{region '#Template'}
	{attribute 'Version' := '1.0.0.0'}
	{attribute 'Tags' := '"LCID": "1031", "Text": "AC, Plant, AHU, Air handling unit"'}
	{attribute 'Tags' := '"LCID": "1033", "Text": "AC, Plant, AHU, Air handling unit"'}
	{attribute 'Description' := '"LCID": "1031", "Text": "Lüftungsanlage"'}
	{attribute 'Description' := '"LCID": "1033", "Text": "Air handling unit"'}
{endregion}
FUNCTION_BLOCK FB_BA_AHU_1St_PrHtr_ErcPl_Col EXTENDS FB_BA_View
VAR_INPUT CONSTANT	
	TOuA					: FB_BA_SensorAnalog_IO;			
	TExhA					: FB_BA_SensorAnalog_IO;	
	TSuA					: FB_BA_SensorAnalog_IO;	
	TExtA					: FB_BA_SensorAnalog_IO;								
	TRm						: FB_BA_SensorAnalog_IO;	
	DiffPrssOuAFilt			: FB_BA_SensorAnalog_IO;											
	FiltOuAMonit			: FB_BA_Hys_21;							
	DiffPrssExtAFilt		: FB_BA_SensorAnalog_IO;				
	FiltExtAMonit			: FB_BA_Hys_21;	
	SumNgtCol				: FB_BA_AC_SumNgtCol;	
	OpMod					: FB_BA_AC_OpMod1St;	
	OuADmp					: FB_BA_Dmp2P;	
	SuAPrss					: FB_BA_SensorAnalog_IO;	
	SuADiffPrss				: FB_BA_SensorAnalog_IO;		
	SuAFan					: FB_BA_MotCtlExt;	
	SuADiffPrssMonit		: FB_BA_FdbAnalog;								
	ExhADmp					: FB_BA_Dmp2P;	
	ExtAPrss				: FB_BA_SensorAnalog_IO;	
	ExtADiffPrss			: FB_BA_SensorAnalog_IO;		
	ExtAFan					: FB_BA_MotCtlExt;								
	ExtADiffPrssMonit		: FB_BA_FdbAnalog;
	SpTRm					: FB_BA_AC_SpTRm_01;	
	TCasCtrl				: FB_BA_AC_TCasCtrl_01;										 								
	TSeqLink				: FB_BA_SequenceLink;
	PreHtr					: FB_BA_AC_PreHtr;	
	Erc						: FB_BA_AC_ErcPl_02;								
	Col						: FB_BA_AC_ColT_02;								
	PlantCtrl				: FB_BA_PlantCtrl;							
	GeneralSettings			: FB_BA_RawSubscriber;
	stGeneralSettings		: ST_BA_GeneralSettings;
END_VAR	
VAR
	PlantLock				: FB_BA_PlantLock	:= (iParent := THIS^);	
	
	PlantControlStatus   	:FB_BA_Label2x :=(iAggregate:=LblControl_PlantControl,		iFunction:=LblFunctions_Status);
	TSequenceControlStatus  :FB_BA_Label2x :=(iAggregate:=LblControl_TSequenceControl,	iFunction:=LblFunctions_Status);	
END_VAR
VAR // added by the converter: edge detectors and wires of the graphical bodies
    _w1 : ANY;
END_VAR

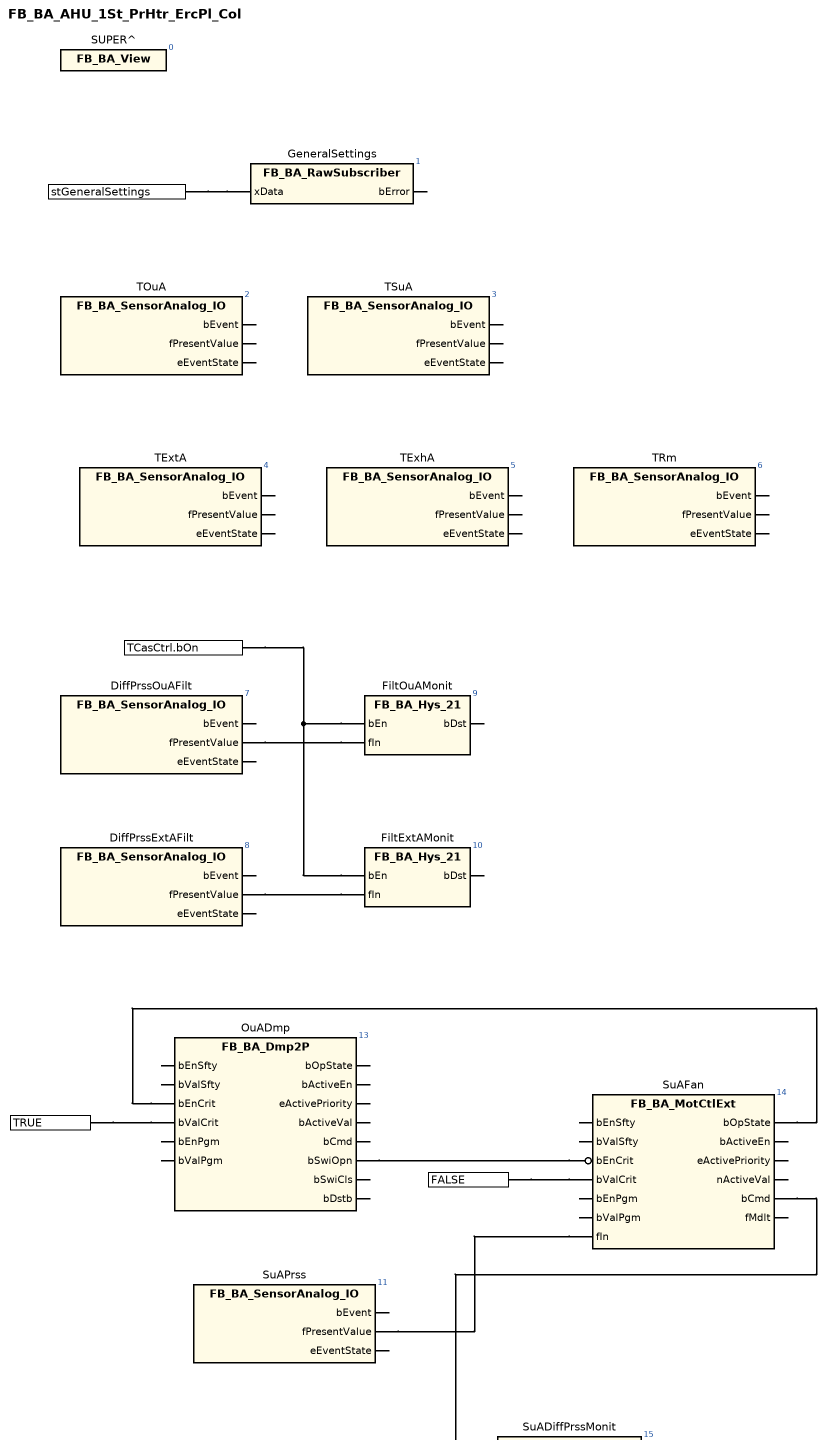
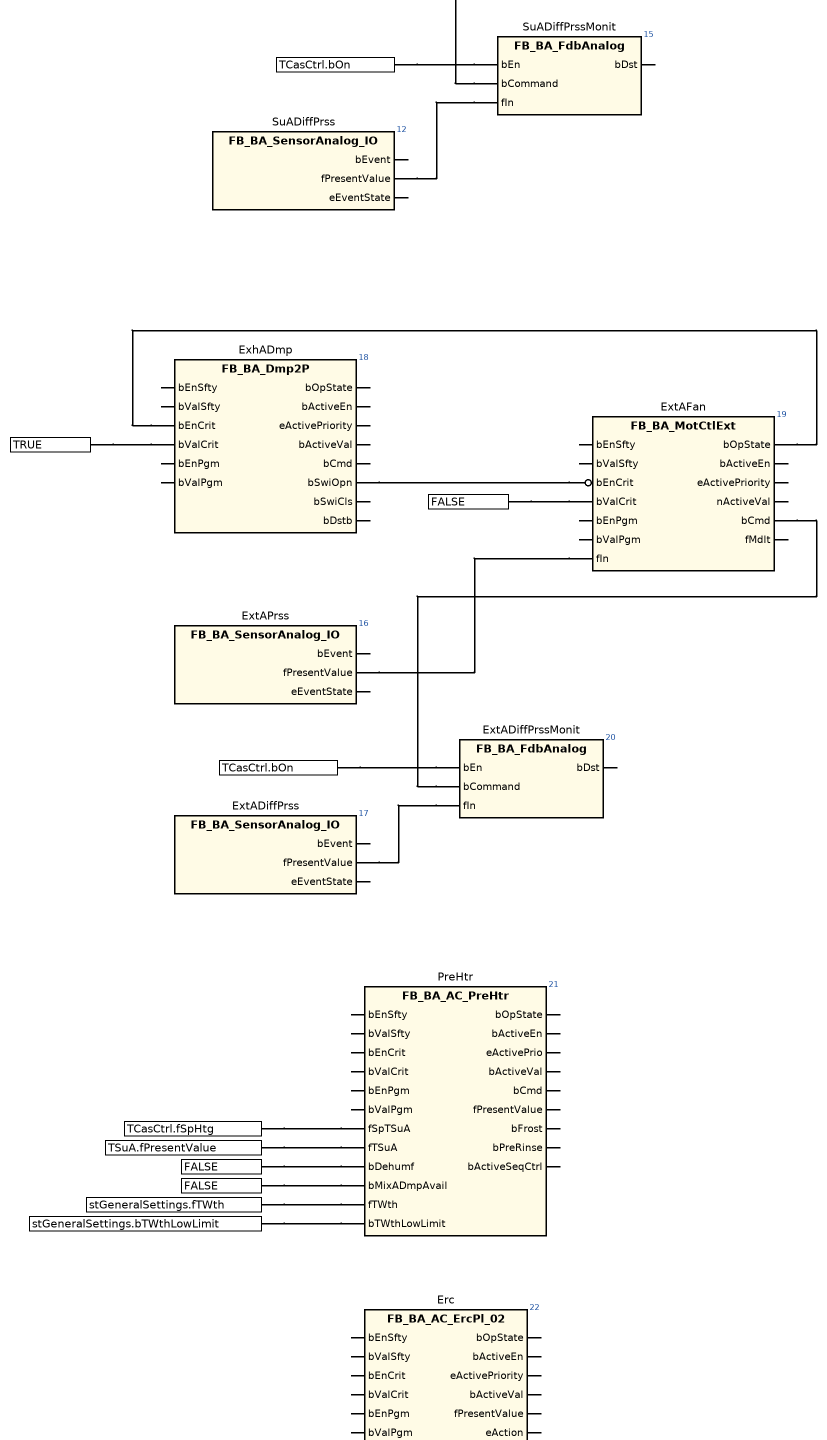
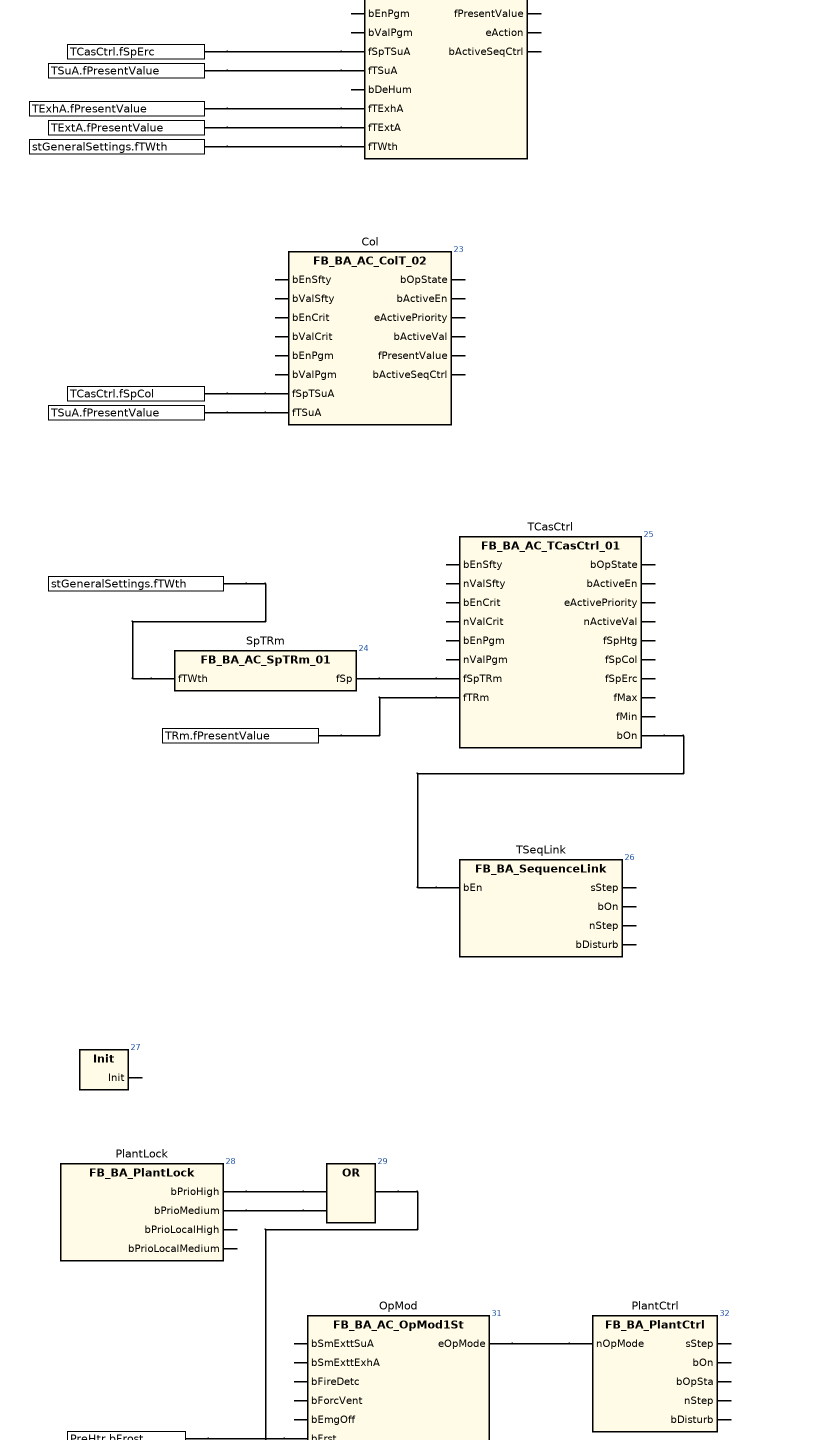
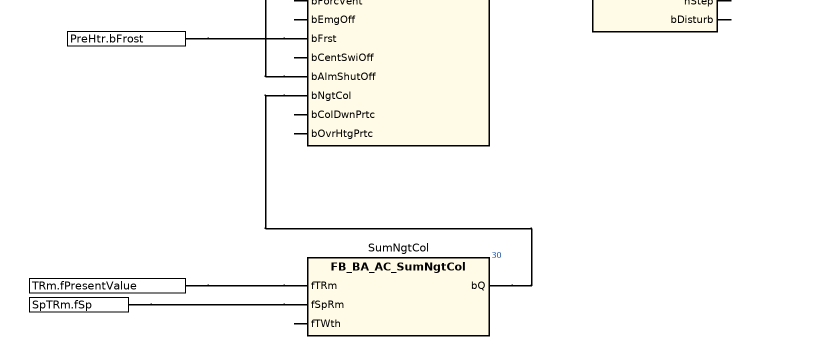
SUPER^(); // FB_BA_View
GeneralSettings(xData := stGeneralSettings); // FB_BA_RawSubscriber
TOuA(); // FB_BA_SensorAnalog_IO
TSuA(); // FB_BA_SensorAnalog_IO
TExtA(); // FB_BA_SensorAnalog_IO
TExhA(); // FB_BA_SensorAnalog_IO
TRm(); // FB_BA_SensorAnalog_IO
DiffPrssOuAFilt(); // FB_BA_SensorAnalog_IO
DiffPrssExtAFilt(); // FB_BA_SensorAnalog_IO
FiltOuAMonit(bEn := TCasCtrl.bOn, fIn := DiffPrssOuAFilt.fPresentValue); // FB_BA_Hys_21
FiltExtAMonit(bEn := TCasCtrl.bOn, fIn := DiffPrssExtAFilt.fPresentValue); // FB_BA_Hys_21
SuAPrss(); // FB_BA_SensorAnalog_IO
SuADiffPrss(); // FB_BA_SensorAnalog_IO
OuADmp(bEnCrit := SuAFan.bOpState, bValCrit := TRUE); // FB_BA_Dmp2P
SuAFan(bEnCrit := NOT OuADmp.bSwiOpn, bValCrit := FALSE, fIn := SuAPrss.fPresentValue); // FB_BA_MotCtlExt
SuADiffPrssMonit(bEn := TCasCtrl.bOn, bCommand := SuAFan.bCmd, fIn := SuADiffPrss.fPresentValue); // FB_BA_FdbAnalog
ExtAPrss(); // FB_BA_SensorAnalog_IO
ExtADiffPrss(); // FB_BA_SensorAnalog_IO
ExhADmp(bEnCrit := ExtAFan.bOpState, bValCrit := TRUE); // FB_BA_Dmp2P
ExtAFan(bEnCrit := NOT ExhADmp.bSwiOpn, bValCrit := FALSE, fIn := ExtAPrss.fPresentValue); // FB_BA_MotCtlExt
ExtADiffPrssMonit(bEn := TCasCtrl.bOn, bCommand := ExtAFan.bCmd, fIn := ExtADiffPrss.fPresentValue); // FB_BA_FdbAnalog
PreHtr(
    fSpTSuA := TCasCtrl.fSpHtg,
    fTSuA := TSuA.fPresentValue,
    bDehumf := FALSE,
    bMixADmpAvail := FALSE,
    fTWth := stGeneralSettings.fTWth,
    bTWthLowLimit := stGeneralSettings.bTWthLowLimit); // FB_BA_AC_PreHtr
Erc(
    fSpTSuA := TCasCtrl.fSpErc,
    fTSuA := TSuA.fPresentValue,
    fTExhA := TExhA.fPresentValue,
    fTExtA := TExtA.fPresentValue,
    fTWth := stGeneralSettings.fTWth); // FB_BA_AC_ErcPl_02
Col(fSpTSuA := TCasCtrl.fSpCol, fTSuA := TSuA.fPresentValue); // FB_BA_AC_ColT_02
SpTRm(fTWth := stGeneralSettings.fTWth); // FB_BA_AC_SpTRm_01
TCasCtrl(fSpTRm := SpTRm.fSp, fTRm := TRm.fPresentValue); // FB_BA_AC_TCasCtrl_01
TSeqLink(bEn := TCasCtrl.bOn); // FB_BA_SequenceLink
Init();
PlantLock(); // FB_BA_PlantLock
_w1 := PlantLock.bPrioHigh OR PlantLock.bPrioMedium;
SumNgtCol(fTRm := TRm.fPresentValue, fSpRm := SpTRm.fSp); // FB_BA_AC_SumNgtCol
OpMod(bFrst := PreHtr.bFrost, bAlmShutOff := _w1, bNgtCol := SumNgtCol.bQ); // FB_BA_AC_OpMod1St
PlantCtrl(nOpMode := OpMod.eOpMode); // FB_BA_PlantCtrl

METHOD FB_init : BOOL
VAR_INPUT
	bInitRetains : BOOL; // if TRUE, the retain variables are initialized (warm start / cold start)
	bInCopyCode : BOOL;  // if TRUE, the instance afterwards gets moved into the copy code (online change)
END_VAR
TOuA.iParent								:= THIS^;		
TOuA.iLabel 								:= LblCmpAC.AHU_TOuA;	
TOuA.sObjectName							:= '{Idx=01}';	
TOuA.eDPADMode								:= E_BA_DPADMode.eInclude;										
TOuA.MV.eUnit								:= E_BA_Unit.eTemperature_DegreesCelsius;
TOuA.MV.fResolution 						:= 0.01;
TOuA.MV.fScaleOffset 						:= 0; 
TOuA.MV.eEnPlantLock						:= E_BA_LockPriority.eNoLock;

TExhA.iParent								:= THIS^;		
TExhA.iLabel 								:= LblCmpAC.AHU_TExhA;	
TExhA.sObjectName							:= '{Idx=01}';												
TExhA.eDPADMode								:= E_BA_DPADMode.eInclude;										
TExhA.MV.eUnit								:= E_BA_Unit.eTemperature_DegreesCelsius;
TExhA.MV.fResolution 						:= 0.01;
TExhA.MV.fScaleOffset 						:= 0; 
TExhA.MV.eEnPlantLock						:= E_BA_LockPriority.eNoLock;

TSuA.iParent								:= THIS^;		
TSuA.iLabel 								:= LblCmpAC.AHU_TSuA;	
TSuA.sObjectName							:= '{Idx=01}';
TSuA.eDPADMode								:= E_BA_DPADMode.eInclude;										
TSuA.MV.eUnit								:= E_BA_Unit.eTemperature_DegreesCelsius;
TSuA.MV.fResolution 						:= 0.01;
TSuA.MV.fScaleOffset 						:= 0; 
TSuA.MV.eEnPlantLock						:= E_BA_LockPriority.eMedium;

TExtA.iParent								:= THIS^;
TExtA.iLabel 								:= LblCmpAC.AHU_TExtA;	
TExtA.sObjectName							:= '{Idx=01}'; 
TExtA.eDPADMode								:= E_BA_DPADMode.eInclude;										
TExtA.MV.eUnit								:= E_BA_Unit.eTemperature_DegreesCelsius;
TExtA.MV.fResolution 						:= 0.01;
TExtA.MV.fScaleOffset 						:= 0; 
TExtA.MV.eEnPlantLock						:= E_BA_LockPriority.eNoLock;

TRm.iParent									:= THIS^;		
TRm.iLabel 									:= LblCmpAC.AHU_TRm;	
TRm.sObjectName								:= '{Idx=01}';
TRm.eDPADMode								:= E_BA_DPADMode.eInclude;										
TRm.MV.eUnit								:= E_BA_Unit.eTemperature_DegreesCelsius;
TRm.MV.fResolution 							:= 0.01;
TRm.MV.fScaleOffset 						:= 0;
TRm.MV.eEnPlantLock							:= E_BA_LockPriority.eNoLock;

DiffPrssOuAFilt.iParent						:= THIS^;		
DiffPrssOuAFilt.iLabel 						:= LblCmpAC.AHU_DiffPrssOuAFilt;	
DiffPrssOuAFilt.sObjectName					:= '{Idx=03}';												
DiffPrssOuAFilt.eDPADMode					:= E_BA_DPADMode.eInclude;										
DiffPrssOuAFilt.MV.eUnit					:= E_BA_Unit.ePressure_Pascals;
DiffPrssOuAFilt.MV.fResolution 				:= 0.03051851;
DiffPrssOuAFilt.MV.fScaleOffset 			:= 0; 
DiffPrssOuAFilt.MV.eEnPlantLock				:= E_BA_LockPriority.eNoLock;

FiltOuAMonit.iParent						:= THIS^;
FiltOuAMonit.iLabel							:= LblCmpAC.AHU_FiltOuAMonit;
FiltOuAMonit.sObjectName					:= '{Idx=01}';										 
FiltOuAMonit.eDPADMode						:= E_BA_DPADMode.eInclude;
FiltOuAMonit.DstPreAlarm.eEnPlantLock		:= E_BA_LockPriority.eNoLock;	
FiltOuAMonit.DstMainAlarm.eEnPlantLock		:= E_BA_LockPriority.eMedium;

DiffPrssExtAFilt.iParent					:= THIS^;		
DiffPrssExtAFilt.iLabel 					:= LblCmpAC.AHU_DiffPrssExtAFilt;	
DiffPrssExtAFilt.sObjectName				:= '{Idx=04}';
DiffPrssExtAFilt.eDPADMode					:= E_BA_DPADMode.eInclude;										
DiffPrssExtAFilt.MV.eUnit					:= E_BA_Unit.ePressure_Pascals;
DiffPrssExtAFilt.MV.fResolution 			:= 0.03051851;
DiffPrssExtAFilt.MV.fScaleOffset 			:= 0; 
DiffPrssExtAFilt.MV.eEnPlantLock			:= E_BA_LockPriority.eNoLock;

FiltExtAMonit.iParent						:= THIS^;
FiltExtAMonit.iLabel						:= LblCmpAC.AHU_FiltExtAMonit;
FiltExtAMonit.sObjectName					:= '{Idx=02}';										 
FiltExtAMonit.eDPADMode						:= E_BA_DPADMode.eInclude;
FiltExtAMonit.DstPreAlarm.eEnPlantLock		:= E_BA_LockPriority.eNoLock;	
FiltExtAMonit.DstMainAlarm.eEnPlantLock		:= E_BA_LockPriority.eMedium;

SumNgtCol.iParent							:= THIS^;
SumNgtCol.iLabel							:= LblCmpAC.AHU_SumNgtCol;
SumNgtCol.sObjectName						:= '{Idx=01}';										 
SumNgtCol.eDPADMode							:= E_BA_DPADMode.eInclude;								

OpMod.iParent								:= THIS^;
OpMod.iLabel								:= LblCmpAC.AHU_OpMod;
OpMod.sObjectName							:= '{Idx=01}';										 
OpMod.eDPADMode								:= E_BA_DPADMode.eInclude;								

OuADmp.iParent								:= THIS^;
OuADmp.iLabel								:= LblCmpAC.AHU_OuADmp;
OuADmp.sObjectName							:= '{Idx=01}';										 
OuADmp.eDPADMode							:= E_BA_DPADMode.eInclude;
OuADmp.MonitOpen.Dst.eEnPlantLock			:= E_BA_LockPriority.eLocalMedium;								
OuADmp.MonitClose.Dst.eEnPlantLock			:= E_BA_LockPriority.eNoLock;								

SuAPrss.iParent								:= THIS^;		
SuAPrss.iLabel 								:= LblCmpAC.AHU_SuAPrss;	
SuAPrss.sObjectName							:= '{Idx=01}';
SuAPrss.eDPADMode							:= E_BA_DPADMode.eInclude;																						
SuAPrss.MV.eUnit							:= E_BA_Unit.ePressure_Pascals;
SuAPrss.MV.fResolution 						:= 0.03051851;
SuAPrss.MV.fScaleOffset 					:= 0;
SuAPrss.MV.eEnPlantLock						:= E_BA_LockPriority.eNoLock;

SuADiffPrss.iParent							:= THIS^;		
SuADiffPrss.iLabel 							:= LblCmpAC.AHU_SuADiffPrss;	
SuADiffPrss.sObjectName						:= '{Idx=01}';
SuADiffPrss.eDPADMode						:= E_BA_DPADMode.eInclude;																						
SuADiffPrss.MV.eUnit						:= E_BA_Unit.ePressure_Pascals;
SuADiffPrss.MV.fResolution 					:= 0.03051851;
SuADiffPrss.MV.fScaleOffset 				:= 0; 
SuADiffPrss.MV.eEnPlantLock					:= E_BA_LockPriority.eNoLock;

SuAFan.iParent								:= THIS^;
SuAFan.iLabel								:= LblCmpAC.AHU_SuAFan;
SuAFan.sObjectName							:= '{Idx=01}';										 
SuAFan.eDPADMode							:= E_BA_DPADMode.eInclude;								
SuAFan.Dst.eEnPlantLock						:= E_BA_LockPriority.eMedium;
SuAFan.ThOvrld.eEnPlantLock					:= E_BA_LockPriority.eMedium;	
SuAFan.MntnSwi.eEnPlantLock					:= E_BA_LockPriority.eMedium;

SuADiffPrssMonit.iParent					:= THIS^;
SuADiffPrssMonit.iLabel						:= LblCmpAC.AHU_SuADiffPrssMonit;
SuADiffPrssMonit.sObjectName				:= '{Idx=01}';										 
SuADiffPrssMonit.eDPADMode					:= E_BA_DPADMode.eInclude;								
SuADiffPrssMonit.Dst.eEnPlantLock			:= E_BA_LockPriority.eMedium;										

ExhADmp.iParent								:= THIS^;
ExhADmp.iLabel								:= LblCmpAC.AHU_ExhADmp;
ExhADmp.sObjectName							:= '{Idx=02}';										 
ExhADmp.eDPADMode							:= E_BA_DPADMode.eInclude;								
ExhADmp.MonitOpen.Dst.eEnPlantLock			:= E_BA_LockPriority.eLocalMedium;								
ExhADmp.MonitClose.Dst.eEnPlantLock			:= E_BA_LockPriority.eNoLock;				

ExtAPrss.iParent							:= THIS^;		
ExtAPrss.iLabel 							:= LblCmpAC.AHU_ExtAPrss;	
ExtAPrss.sObjectName						:= '{Idx=01}';												
ExtAPrss.eDPADMode							:= E_BA_DPADMode.eInclude;																						
ExtAPrss.MV.eUnit							:= E_BA_Unit.ePressure_Pascals;
ExtAPrss.MV.fResolution 					:= 0.03051851;
ExtAPrss.MV.fScaleOffset 					:= 0; 
ExtAPrss.MV.eEnPlantLock					:= E_BA_LockPriority.eNoLock;

ExtADiffPrss.iParent						:= THIS^;		
ExtADiffPrss.iLabel 						:= LblCmpAC.AHU_ExtADiffPrss;	
ExtADiffPrss.sObjectName					:= '{Idx=02}';
ExtADiffPrss.eDPADMode						:= E_BA_DPADMode.eInclude;																						
ExtADiffPrss.MV.eUnit						:= E_BA_Unit.ePressure_Pascals;
ExtADiffPrss.MV.fResolution 				:= 0.03051851;
ExtADiffPrss.MV.fScaleOffset 				:= 0; 
ExtADiffPrss.MV.eEnPlantLock				:= E_BA_LockPriority.eNoLock;

ExtAFan.iParent								:= THIS^;
ExtAFan.iLabel								:= LblCmpAC.AHU_ExtAFan;
ExtAFan.sObjectName							:= '{Idx=01}';										 
ExtAFan.eDPADMode							:= E_BA_DPADMode.eInclude;								
ExtAFan.Dst.eEnPlantLock					:= E_BA_LockPriority.eMedium;
ExtAFan.ThOvrld.eEnPlantLock				:= E_BA_LockPriority.eMedium;	
ExtAFan.MntnSwi.eEnPlantLock				:= E_BA_LockPriority.eMedium;

ExtADiffPrssMonit.iParent					:= THIS^;
ExtADiffPrssMonit.iLabel					:= LblCmpAC.AHU_ExtADiffPrssMonit;
ExtADiffPrssMonit.sObjectName				:= '{Idx=02}';										 
ExtADiffPrssMonit.eDPADMode					:= E_BA_DPADMode.eInclude;								
ExtADiffPrssMonit.Dst.eEnPlantLock			:= E_BA_LockPriority.eMedium;										

SpTRm.iParent								:= THIS^;
SpTRm.iLabel								:= LblCmpAC.AHU_SpTRm;
SpTRm.sObjectName							:= '{Idx=01}';										 
SpTRm.eDPADMode								:= E_BA_DPADMode.eInclude;								

TCasCtrl.iParent							:= THIS^;
TCasCtrl.iLabel								:= LblCmpAC.AHU_TCasCtrl;
TCasCtrl.sObjectName						:= '{Idx=01}';										 
TCasCtrl.eDPADMode							:= E_BA_DPADMode.eInclude;																		 								

TSeqLink.iParent							:= THIS^;
TSeqLink.iLabel								:= LblCmpAC.AHU_TSeqLink;
TSeqLink.sObjectName						:= '{Idx=01,Idx=01}';									
TSeqLink.iReference[1]						:= PreHtr.TSuACtrl.Ctrl;
TSeqLink.iReference[2]						:= Erc.TSuACtrl.Ctrl;
TSeqLink.iReference[3]						:= Col.TSuACtrl.Ctrl;

PreHtr.iParent								:= THIS^;
PreHtr.iLabel								:= LblCmpAC.AHU_PreHtr;
PreHtr.sObjectName							:= '{Idx=01}';										 
PreHtr.eDPADMode							:= E_BA_DPADMode.eIncludeDescription;								
PreHtr.TRt.MV.eEnPlantLock					:= E_BA_LockPriority.eMedium;
PreHtr.TRtCtrl.PreRinseDst.eEnPlantLock		:= E_BA_LockPriority.eNoLock;
PreHtr.TFrost.MV.eEnPlantLock				:= E_BA_LockPriority.eMedium;
PreHtr.FrostThermostat.Input.eEnPlantLock	:= E_BA_LockPriority.eMedium;	
PreHtr.Pu.Dst.eEnPlantLock					:= E_BA_LockPriority.eMedium;

Erc.iParent									:= THIS^;
Erc.iLabel									:= LblCmpAC.AHU_Erc;
Erc.sObjectName								:= '{Idx=01}';										 
Erc.eDPADMode								:= E_BA_DPADMode.eIncludeDescription;																

Col.iParent									:= THIS^;
Col.iLabel									:= LblCmpAC.AHU_Col;
Col.sObjectName								:= '{Idx=01}';										 
Col.eDPADMode								:= E_BA_DPADMode.eIncludeDescription;								

PlantCtrl.iParent							:= THIS^;
PlantCtrl.iLabel							:= LblCmpAC.AHU_PlantCtrl;
PlantCtrl.sObjectName						:= '{Idx=01,Idx=01}';
PlantCtrl.aStateText						:= OpMod.OpModPr.aStateText;	

GeneralSettings.Subject						:= Site.GeneralSettings_Subject;
GeneralSettings.sTarget						:= Site.GeneralSettings_NetId;			
// Die folgenden Aufrufe müssen am Schluss aufgerufen sein!!! // The following calls must be called at the end!!!
PlantCtrl.Clear();
Init_OffOn();
END_METHOD

METHOD Init : BOOL
VAR_INPUT
END_VAR
IF	NOT TSeqLink.bEn
THEN
	TSeqLink.aStateText[1]		:= txtEvent_SupplyAirTControlPeheater;
	TSeqLink.aStateText[2]		:= txtEvent_SupplyAirTControlERC;
	TSeqLink.aStateText[3]		:= txtEvent_SupplyAirTControlCooler;
END_IF
END_METHOD

METHOD Init_OffOn : BOOL

// Betriebsarten der Anlage mit Prioritäten
// plant operations modes with priorities
PlantCtrl.AddOperationMode(nOpMode := E_BA_AC_OpMod01.eOff,							ePrio := E_BA_Priority.eProgram);
PlantCtrl.AddOperationMode(nOpMode := E_BA_AC_OpMod01.eOn,							ePrio := E_BA_Priority.eProgram);
PlantCtrl.AddOperationMode(nOpMode := E_BA_AC_OpMod01.eNightCooling,				ePrio := E_BA_Priority.eProgram);
PlantCtrl.AddOperationMode(nOpMode := E_BA_AC_OpMod01.eCoolDownProtection,			ePrio := E_BA_Priority.eProgram);
PlantCtrl.AddOperationMode(nOpMode := E_BA_AC_OpMod01.eOverHeatingProtection,		ePrio := E_BA_Priority.eProgram);
PlantCtrl.AddOperationMode(nOpMode := E_BA_AC_OpMod01.eFrost,						ePrio := E_BA_Priority.eCritical);
PlantCtrl.AddOperationMode(nOpMode := E_BA_AC_OpMod01.eEmergency,					ePrio := E_BA_Priority.eCritical);
PlantCtrl.AddOperationMode(nOpMode := E_BA_AC_OpMod01.eAlarm,						ePrio := E_BA_Priority.eCritical);
PlantCtrl.AddOperationMode(nOpMode := E_BA_AC_OpMod01.eForcedVentilation,			ePrio := E_BA_Priority.eCritical);
PlantCtrl.AddOperationMode(nOpMode := E_BA_AC_OpMod01.eCentralSwitchOff,			ePrio := E_BA_Priority.eCritical);
PlantCtrl.AddOperationMode(nOpMode := E_BA_AC_OpMod01.eSmokeExtractionProgramm,		ePrio := E_BA_Priority.eLifeSafety);
PlantCtrl.AddOperationMode(nOpMode := E_BA_AC_OpMod01.eSmokeExtractionSupplyAir,	ePrio := E_BA_Priority.eLifeSafety);
PlantCtrl.AddOperationMode(nOpMode := E_BA_AC_OpMod01.eSmokeExtractionExhaustAir,	ePrio := E_BA_Priority.eLifeSafety);
PlantCtrl.AddOperationMode(nOpMode := E_BA_AC_OpMod01.eFire, 						ePrio := E_BA_Priority.eLifeSafety);

// Startsequenz Schrittfolge und Parameter
// Start sequence Step order and parameter
PlantCtrl.AddAggregate(iRef := PreHtr,		bWaitForProcesses := TRUE,	bWaitForEvents := FALSE, tDelayStepDown := T#0S, tDelayStepUp := T#5S);
PlantCtrl.AddAggregate(iRef := OuADmp,		bWaitForProcesses := FALSE, bWaitForEvents := FALSE, tDelayStepDown := T#2S, tDelayStepUp := T#2S);
PlantCtrl.AddAggregate(iRef := ExhADmp,		bWaitForProcesses := FALSE, bWaitForEvents := FALSE, tDelayStepDown := T#2S, tDelayStepUp := T#2S);
PlantCtrl.AddAggregate(iRef := SuAFan,		bWaitForProcesses := FALSE, bWaitForEvents := FALSE, tDelayStepDown := T#2S, tDelayStepUp := T#2S);
PlantCtrl.AddAggregate(iRef := ExtAFan,		bWaitForProcesses := FALSE, bWaitForEvents := FALSE, tDelayStepDown := T#2S, tDelayStepUp := T#2S);
PlantCtrl.AddAggregate(iRef := Erc,			bWaitForProcesses := FALSE, bWaitForEvents := FALSE, tDelayStepDown := T#0S, tDelayStepUp := T#0S);
PlantCtrl.AddAggregate(iRef := Col,			bWaitForProcesses := FALSE, bWaitForEvents := FALSE, tDelayStepDown := T#0S, tDelayStepUp := T#0S);
PlantCtrl.AddAggregate(iRef := TCasCtrl,	bWaitForProcesses := FALSE, bWaitForEvents := FALSE, tDelayStepDown := T#0S, tDelayStepUp := T#0S);

// Aggregatbetriebsarten in Abhängigkeit von den entsprechenden Anlagenbetriebsarten anwenden
// Vorwärmer freigeben in Abhängigkeit von der Anlagenbetriebsart 
// Apply aggregate operation modes dependant on corresponding plant operation modes
// release pre-heater depending on plant operation mode 
PlantCtrl.AssignAggregate1x(nPltOpMode := E_BA_AC_OpMod01.eOff,							iAgg1Ref := PreHtr, nAgg1OpMode := TO_UDINT(FALSE));
PlantCtrl.AssignAggregate1x(nPltOpMode := E_BA_AC_OpMod01.eOn,							iAgg1Ref := PreHtr, nAgg1OpMode := TO_UDINT(TRUE));
PlantCtrl.AssignAggregate1x(nPltOpMode := E_BA_AC_OpMod01.eNightCooling,				iAgg1Ref := PreHtr, nAgg1OpMode := TO_UDINT(FALSE));
PlantCtrl.AssignAggregate1x(nPltOpMode := E_BA_AC_OpMod01.eCoolDownProtection,			iAgg1Ref := PreHtr, nAgg1OpMode := TO_UDINT(TRUE));
PlantCtrl.AssignAggregate1x(nPltOpMode := E_BA_AC_OpMod01.eOverHeatingProtection,		iAgg1Ref := PreHtr, nAgg1OpMode := TO_UDINT(FALSE));
PlantCtrl.AssignAggregate1x(nPltOpMode := E_BA_AC_OpMod01.eFrost,						iAgg1Ref := PreHtr, nAgg1OpMode := TO_UDINT(TRUE));
PlantCtrl.AssignAggregate1x(nPltOpMode := E_BA_AC_OpMod01.eEmergency,					iAgg1Ref := PreHtr, nAgg1OpMode := TO_UDINT(FALSE));
PlantCtrl.AssignAggregate1x(nPltOpMode := E_BA_AC_OpMod01.eAlarm,						iAgg1Ref := PreHtr, nAgg1OpMode := TO_UDINT(FALSE));
PlantCtrl.AssignAggregate1x(nPltOpMode := E_BA_AC_OpMod01.eForcedVentilation,			iAgg1Ref := PreHtr, nAgg1OpMode := TO_UDINT(TRUE));
PlantCtrl.AssignAggregate1x(nPltOpMode := E_BA_AC_OpMod01.eCentralSwitchOff,			iAgg1Ref := PreHtr, nAgg1OpMode := TO_UDINT(FALSE));
PlantCtrl.AssignAggregate1x(nPltOpMode := E_BA_AC_OpMod01.eSmokeExtractionProgramm,		iAgg1Ref := PreHtr, nAgg1OpMode := TO_UDINT(TRUE));
PlantCtrl.AssignAggregate1x(nPltOpMode := E_BA_AC_OpMod01.eSmokeExtractionSupplyAir,	iAgg1Ref := PreHtr, nAgg1OpMode := TO_UDINT(TRUE));
PlantCtrl.AssignAggregate1x(nPltOpMode := E_BA_AC_OpMod01.eSmokeExtractionExhaustAir,	iAgg1Ref := PreHtr, nAgg1OpMode := TO_UDINT(FALSE));
PlantCtrl.AssignAggregate1x(nPltOpMode := E_BA_AC_OpMod01.eFire,						iAgg1Ref := PreHtr, nAgg1OpMode := TO_UDINT(FALSE));

// Aggregatbetriebsarten in Abhängigkeit von den entsprechenden Anlagenbetriebsarten anwenden:
// Erc in Abhängigkeit von der Anlagenbetriebsart freigeben 
// Apply aggregate operation modes dependant on corresponding plant operation modes:
// release Erc depending on plant operation mode 
PlantCtrl.AssignAggregate1x(nPltOpMode := E_BA_AC_OpMod01.eOff,							iAgg1Ref := Erc, nAgg1OpMode := TO_UDINT(FALSE));
PlantCtrl.AssignAggregate1x(nPltOpMode := E_BA_AC_OpMod01.eOn,							iAgg1Ref := Erc, nAgg1OpMode := TO_UDINT(TRUE));
PlantCtrl.AssignAggregate1x(nPltOpMode := E_BA_AC_OpMod01.eNightCooling,				iAgg1Ref := Erc, nAgg1OpMode := TO_UDINT(FALSE));
PlantCtrl.AssignAggregate1x(nPltOpMode := E_BA_AC_OpMod01.eCoolDownProtection,			iAgg1Ref := Erc, nAgg1OpMode := TO_UDINT(TRUE));
PlantCtrl.AssignAggregate1x(nPltOpMode := E_BA_AC_OpMod01.eOverHeatingProtection,		iAgg1Ref := Erc, nAgg1OpMode := TO_UDINT(TRUE));
PlantCtrl.AssignAggregate1x(nPltOpMode := E_BA_AC_OpMod01.eFrost,						iAgg1Ref := Erc, nAgg1OpMode := TO_UDINT(TRUE));
PlantCtrl.AssignAggregate1x(nPltOpMode := E_BA_AC_OpMod01.eEmergency,					iAgg1Ref := Erc, nAgg1OpMode := TO_UDINT(FALSE));
PlantCtrl.AssignAggregate1x(nPltOpMode := E_BA_AC_OpMod01.eAlarm,						iAgg1Ref := Erc, nAgg1OpMode := TO_UDINT(FALSE));
PlantCtrl.AssignAggregate1x(nPltOpMode := E_BA_AC_OpMod01.eForcedVentilation,			iAgg1Ref := Erc, nAgg1OpMode := TO_UDINT(TRUE));
PlantCtrl.AssignAggregate1x(nPltOpMode := E_BA_AC_OpMod01.eCentralSwitchOff,			iAgg1Ref := Erc, nAgg1OpMode := TO_UDINT(FALSE));
PlantCtrl.AssignAggregate1x(nPltOpMode := E_BA_AC_OpMod01.eSmokeExtractionProgramm,		iAgg1Ref := Erc, nAgg1OpMode := TO_UDINT(TRUE));
PlantCtrl.AssignAggregate1x(nPltOpMode := E_BA_AC_OpMod01.eSmokeExtractionSupplyAir,	iAgg1Ref := Erc, nAgg1OpMode := TO_UDINT(TRUE));
PlantCtrl.AssignAggregate1x(nPltOpMode := E_BA_AC_OpMod01.eSmokeExtractionExhaustAir,	iAgg1Ref := Erc, nAgg1OpMode := TO_UDINT(TRUE));
PlantCtrl.AssignAggregate1x(nPltOpMode := E_BA_AC_OpMod01.eFire,						iAgg1Ref := Erc, nAgg1OpMode := TO_UDINT(FALSE));

// Aggregatbetriebsarten in Abhängigkeit von den entsprechenden Anlagenbetriebsarten anwenden:
// Kühler in Abhängigkeit von der Anlagenbetriebsart freigeben
// Apply aggregate operation modes dependant on corresponding plant operation modes:
// release cooler depending on plant operation mode 
PlantCtrl.AssignAggregate1x(nPltOpMode := E_BA_AC_OpMod01.eOff,							iAgg1Ref := Col, nAgg1OpMode := TO_UDINT(FALSE));
PlantCtrl.AssignAggregate1x(nPltOpMode := E_BA_AC_OpMod01.eOn,							iAgg1Ref := Col, nAgg1OpMode := TO_UDINT(TRUE));
PlantCtrl.AssignAggregate1x(nPltOpMode := E_BA_AC_OpMod01.eNightCooling,				iAgg1Ref := Col, nAgg1OpMode := TO_UDINT(FALSE));
PlantCtrl.AssignAggregate1x(nPltOpMode := E_BA_AC_OpMod01.eCoolDownProtection,			iAgg1Ref := Col, nAgg1OpMode := TO_UDINT(FALSE));
PlantCtrl.AssignAggregate1x(nPltOpMode := E_BA_AC_OpMod01.eOverHeatingProtection,		iAgg1Ref := Col, nAgg1OpMode := TO_UDINT(TRUE));
PlantCtrl.AssignAggregate1x(nPltOpMode := E_BA_AC_OpMod01.eFrost,						iAgg1Ref := Col, nAgg1OpMode := TO_UDINT(FALSE));
PlantCtrl.AssignAggregate1x(nPltOpMode := E_BA_AC_OpMod01.eEmergency,					iAgg1Ref := Col, nAgg1OpMode := TO_UDINT(FALSE));
PlantCtrl.AssignAggregate1x(nPltOpMode := E_BA_AC_OpMod01.eAlarm,						iAgg1Ref := Col, nAgg1OpMode := TO_UDINT(FALSE));
PlantCtrl.AssignAggregate1x(nPltOpMode := E_BA_AC_OpMod01.eForcedVentilation,			iAgg1Ref := Col, nAgg1OpMode := TO_UDINT(TRUE));
PlantCtrl.AssignAggregate1x(nPltOpMode := E_BA_AC_OpMod01.eCentralSwitchOff,			iAgg1Ref := Col, nAgg1OpMode := TO_UDINT(FALSE));
PlantCtrl.AssignAggregate1x(nPltOpMode := E_BA_AC_OpMod01.eSmokeExtractionProgramm,		iAgg1Ref := Col, nAgg1OpMode := TO_UDINT(FALSE));
PlantCtrl.AssignAggregate1x(nPltOpMode := E_BA_AC_OpMod01.eSmokeExtractionSupplyAir,	iAgg1Ref := Col, nAgg1OpMode := TO_UDINT(FALSE));
PlantCtrl.AssignAggregate1x(nPltOpMode := E_BA_AC_OpMod01.eSmokeExtractionExhaustAir,	iAgg1Ref := Col, nAgg1OpMode := TO_UDINT(FALSE));
PlantCtrl.AssignAggregate1x(nPltOpMode := E_BA_AC_OpMod01.eFire,						iAgg1Ref := Col, nAgg1OpMode := TO_UDINT(FALSE));

// Aggregatbetriebsarten in Abhängigkeit von den entsprechenden Anlagenbetriebsarten anwenden:
// Außenluftklappe freigeben in Abhängigkeit von der Anlagenbetriebsart 
// Apply aggregate operation modes dependant on corresponding plant operation modes:
// release outside air damper depending on plant operation mode 
PlantCtrl.AssignAggregate1x(nPltOpMode := E_BA_AC_OpMod01.eOff,							iAgg1Ref := OuADmp, nAgg1OpMode := TO_UDINT(FALSE));
PlantCtrl.AssignAggregate1x(nPltOpMode := E_BA_AC_OpMod01.eOn,							iAgg1Ref := OuADmp, nAgg1OpMode := TO_UDINT(TRUE));
PlantCtrl.AssignAggregate1x(nPltOpMode := E_BA_AC_OpMod01.eNightCooling,				iAgg1Ref := OuADmp, nAgg1OpMode := TO_UDINT(TRUE));
PlantCtrl.AssignAggregate1x(nPltOpMode := E_BA_AC_OpMod01.eCoolDownProtection,			iAgg1Ref := OuADmp, nAgg1OpMode := TO_UDINT(TRUE));
PlantCtrl.AssignAggregate1x(nPltOpMode := E_BA_AC_OpMod01.eOverHeatingProtection,		iAgg1Ref := OuADmp, nAgg1OpMode := TO_UDINT(TRUE));
PlantCtrl.AssignAggregate1x(nPltOpMode := E_BA_AC_OpMod01.eFrost,						iAgg1Ref := OuADmp, nAgg1OpMode := TO_UDINT(FALSE));
PlantCtrl.AssignAggregate1x(nPltOpMode := E_BA_AC_OpMod01.eEmergency,					iAgg1Ref := OuADmp, nAgg1OpMode := TO_UDINT(FALSE));
PlantCtrl.AssignAggregate1x(nPltOpMode := E_BA_AC_OpMod01.eAlarm,						iAgg1Ref := OuADmp, nAgg1OpMode := TO_UDINT(FALSE));
PlantCtrl.AssignAggregate1x(nPltOpMode := E_BA_AC_OpMod01.eForcedVentilation,			iAgg1Ref := OuADmp, nAgg1OpMode := TO_UDINT(TRUE));
PlantCtrl.AssignAggregate1x(nPltOpMode := E_BA_AC_OpMod01.eCentralSwitchOff,			iAgg1Ref := OuADmp, nAgg1OpMode := TO_UDINT(FALSE));
PlantCtrl.AssignAggregate1x(nPltOpMode := E_BA_AC_OpMod01.eSmokeExtractionProgramm,		iAgg1Ref := OuADmp, nAgg1OpMode := TO_UDINT(TRUE));
PlantCtrl.AssignAggregate1x(nPltOpMode := E_BA_AC_OpMod01.eSmokeExtractionSupplyAir,	iAgg1Ref := OuADmp, nAgg1OpMode := TO_UDINT(TRUE));
PlantCtrl.AssignAggregate1x(nPltOpMode := E_BA_AC_OpMod01.eSmokeExtractionExhaustAir,	iAgg1Ref := OuADmp, nAgg1OpMode := TO_UDINT(FALSE));
PlantCtrl.AssignAggregate1x(nPltOpMode := E_BA_AC_OpMod01.eFire,						iAgg1Ref := OuADmp, nAgg1OpMode := TO_UDINT(FALSE));

// Aggregatbetriebsarten in Abhängigkeit von den entsprechenden Anlagenbetriebsarten anwenden:
// Zuluftventilator freigeben in Abhängigkeit von der Anlagenbetriebsart 
// Apply aggregate operation modes dependant on corresponding plant operation modes:
// release supply air fan depending on plant operation mode 
PlantCtrl.AssignAggregate1x(nPltOpMode := E_BA_AC_OpMod01.eOff,							iAgg1Ref := SuAFan, nAgg1OpMode := E_BA_MdltCmd.eOff);
PlantCtrl.AssignAggregate1x(nPltOpMode := E_BA_AC_OpMod01.eOn,							iAgg1Ref := SuAFan, nAgg1OpMode := E_BA_MdltCmd.eOn);
PlantCtrl.AssignAggregate1x(nPltOpMode := E_BA_AC_OpMod01.eNightCooling,				iAgg1Ref := SuAFan, nAgg1OpMode := E_BA_MdltCmd.eOn);
PlantCtrl.AssignAggregate1x(nPltOpMode := E_BA_AC_OpMod01.eCoolDownProtection,			iAgg1Ref := SuAFan, nAgg1OpMode := E_BA_MdltCmd.eOn);
PlantCtrl.AssignAggregate1x(nPltOpMode := E_BA_AC_OpMod01.eOverHeatingProtection,		iAgg1Ref := SuAFan, nAgg1OpMode := E_BA_MdltCmd.eOn);
PlantCtrl.AssignAggregate1x(nPltOpMode := E_BA_AC_OpMod01.eFrost,						iAgg1Ref := SuAFan, nAgg1OpMode := E_BA_MdltCmd.eOff);
PlantCtrl.AssignAggregate1x(nPltOpMode := E_BA_AC_OpMod01.eEmergency,					iAgg1Ref := SuAFan, nAgg1OpMode := E_BA_MdltCmd.eOff);
PlantCtrl.AssignAggregate1x(nPltOpMode := E_BA_AC_OpMod01.eAlarm,						iAgg1Ref := SuAFan, nAgg1OpMode := E_BA_MdltCmd.eOff);
PlantCtrl.AssignAggregate1x(nPltOpMode := E_BA_AC_OpMod01.eForcedVentilation,			iAgg1Ref := SuAFan, nAgg1OpMode := E_BA_MdltCmd.eOn);
PlantCtrl.AssignAggregate1x(nPltOpMode := E_BA_AC_OpMod01.eCentralSwitchOff,			iAgg1Ref := SuAFan, nAgg1OpMode := E_BA_MdltCmd.eOff);
PlantCtrl.AssignAggregate1x(nPltOpMode := E_BA_AC_OpMod01.eSmokeExtractionProgramm,		iAgg1Ref := SuAFan, nAgg1OpMode := E_BA_MdltCmd.eOn);
PlantCtrl.AssignAggregate1x(nPltOpMode := E_BA_AC_OpMod01.eSmokeExtractionSupplyAir,	iAgg1Ref := SuAFan, nAgg1OpMode := E_BA_MdltCmd.eOn);
PlantCtrl.AssignAggregate1x(nPltOpMode := E_BA_AC_OpMod01.eSmokeExtractionExhaustAir,	iAgg1Ref := SuAFan, nAgg1OpMode := E_BA_MdltCmd.eOff);
PlantCtrl.AssignAggregate1x(nPltOpMode := E_BA_AC_OpMod01.eFire,						iAgg1Ref := SuAFan, nAgg1OpMode := E_BA_MdltCmd.eOff);

// Aggregatbetriebsarten in Abhängigkeit von den entsprechenden Anlagenbetriebsarten anwenden:
// Fortluftklappe freigeben in Abhängigkeit von der Anlagenbetriebsart 
// Apply aggregate operation modes dependant on corresponding plant operation modes:
// release exhaust air damper depending on plant operation mode 
PlantCtrl.AssignAggregate1x(nPltOpMode := E_BA_AC_OpMod01.eOff,							iAgg1Ref := ExhADmp, nAgg1OpMode := TO_UDINT(FALSE));
PlantCtrl.AssignAggregate1x(nPltOpMode := E_BA_AC_OpMod01.eOn,							iAgg1Ref := ExhADmp, nAgg1OpMode := TO_UDINT(TRUE));
PlantCtrl.AssignAggregate1x(nPltOpMode := E_BA_AC_OpMod01.eNightCooling,				iAgg1Ref := ExhADmp, nAgg1OpMode := TO_UDINT(TRUE));
PlantCtrl.AssignAggregate1x(nPltOpMode := E_BA_AC_OpMod01.eCoolDownProtection,			iAgg1Ref := ExhADmp, nAgg1OpMode := TO_UDINT(TRUE));
PlantCtrl.AssignAggregate1x(nPltOpMode := E_BA_AC_OpMod01.eOverHeatingProtection,		iAgg1Ref := ExhADmp, nAgg1OpMode := TO_UDINT(TRUE));
PlantCtrl.AssignAggregate1x(nPltOpMode := E_BA_AC_OpMod01.eFrost,						iAgg1Ref := ExhADmp, nAgg1OpMode := TO_UDINT(FALSE));
PlantCtrl.AssignAggregate1x(nPltOpMode := E_BA_AC_OpMod01.eEmergency,					iAgg1Ref := ExhADmp, nAgg1OpMode := TO_UDINT(FALSE));
PlantCtrl.AssignAggregate1x(nPltOpMode := E_BA_AC_OpMod01.eAlarm,						iAgg1Ref := ExhADmp, nAgg1OpMode := TO_UDINT(FALSE));
PlantCtrl.AssignAggregate1x(nPltOpMode := E_BA_AC_OpMod01.eForcedVentilation,			iAgg1Ref := ExhADmp, nAgg1OpMode := TO_UDINT(TRUE));
PlantCtrl.AssignAggregate1x(nPltOpMode := E_BA_AC_OpMod01.eCentralSwitchOff,			iAgg1Ref := ExhADmp, nAgg1OpMode := TO_UDINT(FALSE));
PlantCtrl.AssignAggregate1x(nPltOpMode := E_BA_AC_OpMod01.eSmokeExtractionProgramm,		iAgg1Ref := ExhADmp, nAgg1OpMode := TO_UDINT(TRUE));
PlantCtrl.AssignAggregate1x(nPltOpMode := E_BA_AC_OpMod01.eSmokeExtractionSupplyAir,	iAgg1Ref := ExhADmp, nAgg1OpMode := TO_UDINT(FALSE));
PlantCtrl.AssignAggregate1x(nPltOpMode := E_BA_AC_OpMod01.eSmokeExtractionExhaustAir,	iAgg1Ref := ExhADmp, nAgg1OpMode := TO_UDINT(TRUE));
PlantCtrl.AssignAggregate1x(nPltOpMode := E_BA_AC_OpMod01.eFire,						iAgg1Ref := ExhADmp, nAgg1OpMode := TO_UDINT(FALSE));

// Aggregatbetriebsarten in Abhängigkeit von den entsprechenden Anlagenbetriebsarten anwenden:
// Abluftventilator freigeben in Abhängigkeit von der Anlagenbetriebsart 
// Apply aggregate operation modes dependant on corresponding plant operation modes:
// release extract air fan depending on plant operation mode 
PlantCtrl.AssignAggregate1x(nPltOpMode := E_BA_AC_OpMod01.eOff,							iAgg1Ref := ExtAFan, nAgg1OpMode := E_BA_MdltCmd.eOff);
PlantCtrl.AssignAggregate1x(nPltOpMode := E_BA_AC_OpMod01.eOn,							iAgg1Ref := ExtAFan, nAgg1OpMode := E_BA_MdltCmd.eOn); 
PlantCtrl.AssignAggregate1x(nPltOpMode := E_BA_AC_OpMod01.eNightCooling,				iAgg1Ref := ExtAFan, nAgg1OpMode := E_BA_MdltCmd.eOn); 
PlantCtrl.AssignAggregate1x(nPltOpMode := E_BA_AC_OpMod01.eCoolDownProtection,			iAgg1Ref := ExtAFan, nAgg1OpMode := E_BA_MdltCmd.eOn); 
PlantCtrl.AssignAggregate1x(nPltOpMode := E_BA_AC_OpMod01.eOverHeatingProtection,		iAgg1Ref := ExtAFan, nAgg1OpMode := E_BA_MdltCmd.eOn); 
PlantCtrl.AssignAggregate1x(nPltOpMode := E_BA_AC_OpMod01.eFrost,						iAgg1Ref := ExtAFan, nAgg1OpMode := E_BA_MdltCmd.eOff);
PlantCtrl.AssignAggregate1x(nPltOpMode := E_BA_AC_OpMod01.eEmergency,					iAgg1Ref := ExtAFan, nAgg1OpMode := E_BA_MdltCmd.eOff);
PlantCtrl.AssignAggregate1x(nPltOpMode := E_BA_AC_OpMod01.eAlarm,						iAgg1Ref := ExtAFan, nAgg1OpMode := E_BA_MdltCmd.eOff);
PlantCtrl.AssignAggregate1x(nPltOpMode := E_BA_AC_OpMod01.eForcedVentilation,			iAgg1Ref := ExtAFan, nAgg1OpMode := E_BA_MdltCmd.eOn); 
PlantCtrl.AssignAggregate1x(nPltOpMode := E_BA_AC_OpMod01.eCentralSwitchOff,			iAgg1Ref := ExtAFan, nAgg1OpMode := E_BA_MdltCmd.eOff);
PlantCtrl.AssignAggregate1x(nPltOpMode := E_BA_AC_OpMod01.eSmokeExtractionProgramm,		iAgg1Ref := ExtAFan, nAgg1OpMode := E_BA_MdltCmd.eOn); 
PlantCtrl.AssignAggregate1x(nPltOpMode := E_BA_AC_OpMod01.eSmokeExtractionSupplyAir,	iAgg1Ref := ExtAFan, nAgg1OpMode := E_BA_MdltCmd.eOff);
PlantCtrl.AssignAggregate1x(nPltOpMode := E_BA_AC_OpMod01.eSmokeExtractionExhaustAir,	iAgg1Ref := ExtAFan, nAgg1OpMode := E_BA_MdltCmd.eOn); 
PlantCtrl.AssignAggregate1x(nPltOpMode := E_BA_AC_OpMod01.eFire,						iAgg1Ref := ExtAFan, nAgg1OpMode := E_BA_MdltCmd.eOff);

// Aggregatbetriebsarten in Abhängigkeit von den entsprechenden Anlagenbetriebsarten anwenden:
// Kaskadenregelung freigeben in Abhängigkeit von der Anlagenbetriebsart 
// Apply aggregate operation modes dependant on corresponding plant operation modes:
// release cascade control depending on plant operation mode 
PlantCtrl.AssignAggregate1x(nPltOpMode := E_BA_AC_OpMod01.eOff,							iAgg1Ref := TCasCtrl, nAgg1OpMode := E_BA_MdltCmd.eOff);
PlantCtrl.AssignAggregate1x(nPltOpMode := E_BA_AC_OpMod01.eOn,							iAgg1Ref := TCasCtrl, nAgg1OpMode := E_BA_MdltCmd.eOn);
PlantCtrl.AssignAggregate1x(nPltOpMode := E_BA_AC_OpMod01.eNightCooling,				iAgg1Ref := TCasCtrl, nAgg1OpMode := E_BA_MdltCmd.eOff);
PlantCtrl.AssignAggregate1x(nPltOpMode := E_BA_AC_OpMod01.eCoolDownProtection,			iAgg1Ref := TCasCtrl, nAgg1OpMode := E_BA_MdltCmd.eMax);
PlantCtrl.AssignAggregate1x(nPltOpMode := E_BA_AC_OpMod01.eOverHeatingProtection,		iAgg1Ref := TCasCtrl, nAgg1OpMode := E_BA_MdltCmd.eMin);
PlantCtrl.AssignAggregate1x(nPltOpMode := E_BA_AC_OpMod01.eFrost,						iAgg1Ref := TCasCtrl, nAgg1OpMode := E_BA_MdltCmd.eOff);
PlantCtrl.AssignAggregate1x(nPltOpMode := E_BA_AC_OpMod01.eEmergency,					iAgg1Ref := TCasCtrl, nAgg1OpMode := E_BA_MdltCmd.eOff);
PlantCtrl.AssignAggregate1x(nPltOpMode := E_BA_AC_OpMod01.eAlarm,						iAgg1Ref := TCasCtrl, nAgg1OpMode := E_BA_MdltCmd.eOff);
PlantCtrl.AssignAggregate1x(nPltOpMode := E_BA_AC_OpMod01.eForcedVentilation,			iAgg1Ref := TCasCtrl, nAgg1OpMode := E_BA_MdltCmd.eOn);
PlantCtrl.AssignAggregate1x(nPltOpMode := E_BA_AC_OpMod01.eCentralSwitchOff,			iAgg1Ref := TCasCtrl, nAgg1OpMode := E_BA_MdltCmd.eMin);
PlantCtrl.AssignAggregate1x(nPltOpMode := E_BA_AC_OpMod01.eSmokeExtractionProgramm,		iAgg1Ref := TCasCtrl, nAgg1OpMode := E_BA_MdltCmd.eMin);
PlantCtrl.AssignAggregate1x(nPltOpMode := E_BA_AC_OpMod01.eSmokeExtractionSupplyAir,	iAgg1Ref := TCasCtrl, nAgg1OpMode := E_BA_MdltCmd.eMin);
PlantCtrl.AssignAggregate1x(nPltOpMode := E_BA_AC_OpMod01.eSmokeExtractionExhaustAir,	iAgg1Ref := TCasCtrl, nAgg1OpMode := E_BA_MdltCmd.eOff);
PlantCtrl.AssignAggregate1x(nPltOpMode := E_BA_AC_OpMod01.eFire,						iAgg1Ref := TCasCtrl, nAgg1OpMode := E_BA_MdltCmd.eOff);
END_METHOD

END_FUNCTION_BLOCK

(* stored: Version 1.1.0.1, ProductVersion 3.1.4024.9
   POU FB_BA_AHU_1St_PrHtr_ErcPl_Col: Id {3ab6c3f6-1500-4003-b83a-8b5bef71ccad}, SpecialFunc None
   Folder Initialization: Id {a172b826-54c6-42f9-b2aa-ced024f6e23f}
   Method FB_init: Id {117b0697-8883-45fa-9f9c-d79a25fd0d56}
   Method Init: Id {8f15b6f5-7aae-4f40-8890-2e283c77e35d}
   Method Init_OffOn: Id {da1fac7c-7cd4-47be-b06a-9e5fccfa1a9c} *)
